// TwinCAT 3 PLC project RT1
// ProgramVersion: 3.1.4023.0
// libraries:
//   Tc2_Standard, * (Beckhoff Automation GmbH)
//   Tc2_System, * (Beckhoff Automation GmbH)
//   Tc2_Utilities, * (Beckhoff Automation GmbH)
//   Tc3_IotBase, * (Beckhoff Automation GmbH)
//   Tc3_JsonXml, * (Beckhoff Automation GmbH)
//   Tc3_Module, * (Beckhoff Automation GmbH)
// project tree:
//   DUTs/ stValues.TcDUT
//   / PlcTask.TcTTO
//   POUs/ FB_MQTT.TcPOU, MAIN.TcPOU
// real-time tasks:
//   TASK PlcTask: cycle T#10ms, priority 20, ADS port 350

CONFIGURATION RT1
    RESOURCE PLC ON TwinCAT3
        TASK PlcTask(INTERVAL := T#10ms, PRIORITY := 20);
        PROGRAM MAIN WITH PlcTask : MAIN;
    END_RESOURCE
END_CONFIGURATION

// ---- DUTs/stValues.TcDUT
TYPE stValues :
STRUCT
	Sensor1:REAL;
	Sensor2:UDINT;
	Sensor3:UDINT;
END_STRUCT
END_TYPE

// ---- POUs/MAIN.TcPOU
PROGRAM MAIN
VAR
	cliente:FB_IotMqttClient;	//Efetivamente o cliente MQTT
	bInit: BOOL:=TRUE;
	bConnect: BOOL;
	sTopicPub:STRING(255):='Topic01';
	sPayloadPub:STRING(255);

	
	i: INT;
	asTopicSub: ARRAY [1..3] OF STRING := ['Topic01', 'Maq/Sensores', 'Maq/Prod'];
	fbMessage: FB_IotMqttMessage;
	bPublish: BOOL;
	
	valoresEnviar: stValues := (Sensor1 := 25.4, Sensor2 := 32, Sensor3 := 64);
	timeHand:FB_LocalSystemTime;
	fbJson:FB_JsonSaxWriter;
	fbJsonDataType:FB_JsonReadWriteDatatype;
	sJsonDoc:STRING(255);
	sJsonDoc2:STRING(2000);
	symbolReturn:stValues;
	bConvertBack: BOOL;
	sensores: stSensores := (bSensor1 := TRUE, rTemp01 := 36.7, rTemp02 := 123.87, udiValor := 32);
	prod: stProducao := (iQdtProd := 123, iQualidade := 321, iPcPerDay := 475);
	sTopicSensores:STRING:='Maq/Sensores';
	sTopicProd:STRING:='Maq/Prod';
	bPublishSensores,bPublishProd:BOOL;
END_VAR

IF bInit THEN
	bInit:=FALSE;
	cliente.sClientId:='Test01';
	cliente.sHostName:='localhost';
	cliente.nHostPort:=1883;
	cliente.ipMessageQueue:=messaQueue;
END_IF

cliente.Execute(bConnect);

IF cliente.bConnected THEN
	FOR i:=1 TO 3 DO
		IF abSubscribe[i] AND NOT abSubscribed[i] THEN
			abSubscribed[i]:=cliente.Subscribe(sTopic:=asTopicSub[i],eQoS:=TcIotMqttQos.AtMostOnceDelivery);
		END_IF
	END_FOR
	IF bPublish THEN
		fbJson.ResetDocument();
		fbJsonDataType.AddJsonValueFromSymbol(fbJson,'stValues',SIZEOF(valoresEnviar),ADR(valoresEnviar));
		sJsonDoc:=fbJson.GetDocument();
		fbJson.CopyDocument(sJsonDoc2,SIZEOF(sJsonDoc2));

		cliente.Publish(sTopic:= sTopicPub, 
		pPayload:= ADR(sJsonDoc2), nPayloadSize:= LEN2(ADR(sJsonDoc2))+1, 
		eQoS:= TcIotMqttQos.AtMostOnceDelivery, bRetain:= FALSE, bQueue:= FALSE );
		bPublish:=FALSE;
	END_IF
	
	IF bPublishSensores THEN
		fbJson.ResetDocument();
		fbJsonDataType.AddJsonValueFromSymbol(fbJson,'stValues',SIZEOF(valoresEnviar),ADR(valoresEnviar));
		sJsonDoc:=fbJson.GetDocument();
		fbJson.CopyDocument(sJsonDoc2,SIZEOF(sJsonDoc2));

		cliente.Publish(sTopic:=sTopicSensores,
		pPayload:= ADR(sJsonDoc2), nPayloadSize:= LEN2(ADR(sJsonDoc2))+1, 
		eQoS:= TcIotMqttQos.AtMostOnceDelivery, bRetain:= FALSE, bQueue:= FALSE );
		bPublishSensores:=FALSE;
	END_IF
	
	IF bPublishProd THEN
		fbJson.ResetDocument();
		fbJsonDataType.AddJsonValueFromSymbol(fbJson,'stProducao',SIZEOF(prod),ADR(prod));
		sJsonDoc:=fbJson.GetDocument();
		fbJson.CopyDocument(sJsonDoc2,SIZEOF(sJsonDoc2));

		cliente.Publish(sTopic:=sTopicProd,
		pPayload:= ADR(sJsonDoc2), nPayloadSize:= LEN2(ADR(sJsonDoc2))+1, 
		eQoS:= TcIotMqttQos.AtMostOnceDelivery, bRetain:= FALSE, bQueue:= FALSE );		
		bPublishProd:=FALSE;
	END_IF
END_IF

IF bConvertBack THEN
	fbJsonDataType.SetSymbolFromJson(sJsonDoc2,'stValues',SIZEOF(symbolReturn),ADR(symbolReturn));
END_IF

END_PROGRAM

// ---- POUs/FB_MQTT.TcPOU
FUNCTION_BLOCK FB_MQTT
VAR_INPUT	
	bConnect : BOOL; // Flag de conexão, inicia conexão
	bPublish : BOOL; // Flag para autorizar publicação
	iDataQtd : INT;  // Quantidade de variáveis para transmitir (Unitário)
	valoresEnviar : stValues; // Valores para enviar
END_VAR
VAR_OUTPUT
END_VAR
VAR
	bInit		: BOOL;
	Client		: FB_IotMqttClient;
	i			: INT;
	messaQueue	: I_IotMqttMessageQueue;
	
	abSubscribe		: ARRAY[1..iDataQtd] OF BOOL;
	abSubscribed	: ARRAY[1..iDataQtd] OF BOOL;
	asTopicSub		: STRING;
	
	fbJson			: FB_JsonSaxWriter;
	fbJsonDataType  : FB_JsonReadWriteDatatype;
END_VAR

IF bInit THEN
	bInit:=FALSE;
	Client.sClientId:='Test01';
	Client.sHostName:='localhost';
	Client.nHostPort:=1883;
	Client.ipMessageQueue:=messaQueue;
END_IF

Client.Execute(bConnect);

IF Client.bConnected THEN
	FOR i:=1 TO 3 DO
		IF abSubscribe[i] AND NOT abSubscribed[i] THEN
			abSubscribed[i]:=Client.Subscribe(sTopic:=asTopicSub[i],eQoS:=TcIotMqttQos.AtMostOnceDelivery);
		END_IF
	END_FOR
	IF bPublish THEN
		fbJson.ResetDocument();
		fbJsonDataType.AddJsonValueFromSymbol(fbJson,'stValues',SIZEOF(valoresEnviar),ADR(valoresEnviar));
		sJsonDoc:=fbJson.GetDocument();
		fbJson.CopyDocument(sJsonDoc2,SIZEOF(sJsonDoc2));

		cliente.Publish(sTopic:= sTopicPub, 
		pPayload:= ADR(sJsonDoc2), nPayloadSize:= LEN2(ADR(sJsonDoc2))+1, 
		eQoS:= TcIotMqttQos.AtMostOnceDelivery, bRetain:= FALSE, bQueue:= FALSE );
		bPublish:=FALSE;
	END_IF

END_FUNCTION_BLOCK
